(* PLC project Generated.project, CODESYS CODESYS V3.5 SP19 Patch 1 *)
(* stored: creationDateTime 2026-09-06T13:00:42.500763, modificationDateTime 2026-09-06T13:00:42.500763 *)

TYPE ST_Chain_Translation_Outputs : STRUCT
  Idx501_CmdDriveControlWord : WORD;  (* Mot de Commande Transmis EtherCAT AC600 *)
  Idx502_CmdDriveFreq_Hz : UINT;  (* [0.01Hz] Consigne Fréquence Transmise EtherCAT *)
  Idx503_CmdBrakeRelease_RQ : BOOL;  (* 1 = Bobine Frein Translation Alimentée (Ouvert) *)
END_STRUCT;
END_TYPE
